// TIA Portal V17 program export: 1 tag tables, 0 data types, 3 data blocks, 1 code blocks (in call order from the OBs), 3 instance data blocks

VAR_GLOBAL   // PLC tag table "Default tag table"
   Batch_WeightScale_Done AT %M2.2 : Bool;
   Batch_FillToMixer_Done AT %M2.3 : Bool;
   Batch_Mixing_Done AT %M2.4 : Bool;
   Batch_Fillto_Pasteurisation_Done AT %M2.5 : Bool;
   Batch_Pasteurizing_Done AT %M2.6 : Bool;
   Filler_Ready AT %M2.7 : Bool;
   Clock_Byte AT %MB0 : Byte;
   Clock_10Hz AT %M0.0 : Bool;
   Clock_5Hz AT %M0.1 : Bool;
   "Clock_2.5Hz" AT %M0.2 : Bool;
   Clock_2Hz AT %M0.3 : Bool;
   "Clock_1.25Hz" AT %M0.4 : Bool;
   Clock_1Hz AT %M0.5 : Bool;
   "Clock_0.625Hz" AT %M0.6 : Bool;
   "Clock_0.5Hz" AT %M0.7 : Bool;
END_VAR

DATA_BLOCK "Device"   // DB1
{ S7_Optimized_Access := 'FALSE' }
VERSION : 0.1
// stored: AutoNumber true, DBAccessibleFromOPCUA true, DBAccessibleFromWebserver true, IsOnlyStoredInLoadMemory false, IsWriteProtectedInAS false
   VAR
      V1103 : Bool;
      V01101 : Bool;
      V2101 : Bool;
      V3101 : Bool;
      V1102 : Bool;
      V2102 : Bool;
      V3102 : Bool;
      V4101 : Bool;
      V4102 : Bool;
      V4103 : Bool;
      W1111 : Real;
      W2111 : Real;
      W3111 : Real;
      L4141 : Real;
      AGR5101 : Bool;
      PUMP4121 : Bool;
      PASTEURISING_MACHINE_ON : Bool;
      FILLING_MACHINE : Bool;
      V1101 : Bool;
      L5141 : Real;
      V01101_s : Bool;
      V2101_s : Bool;
      V3101_s : Bool;
      V1102_s : Bool;
      V2102_s : Bool;
      V3102_s : Bool;
      AGR5101_s : Bool;
      V4101_s : Bool;
      PUMP4121_s : Bool;
      V4102_s : Bool;
      PASTEURISING_MACHINE_ON_s : Bool;
      FILLING_MACHINE_s : Bool;
      V2102_ss : Bool;
      V4103_s : Bool;
   END_VAR
BEGIN
END_DATA_BLOCK

DATA_BLOCK "Recipe_Parameter"   // DB2
{ S7_Optimized_Access := 'FALSE' }
VERSION : 0.1
// stored: AutoNumber true, DBAccessibleFromOPCUA true, DBAccessibleFromWebserver true, IsOnlyStoredInLoadMemory false, IsWriteProtectedInAS false
   VAR
      SelectedFlavor : Int;
      Milk_Volume : Real;
      Flavor_Volume : Real;
      Mixing_Time : Time;
      Pasteurising_Time : Time;
   END_VAR
BEGIN
END_DATA_BLOCK

DATA_BLOCK "SCADA"   // DB3
{ S7_Optimized_Access := 'FALSE' }
VERSION : 0.1
// stored: AutoNumber true, DBAccessibleFromOPCUA true, DBAccessibleFromWebserver true, IsOnlyStoredInLoadMemory false, IsWriteProtectedInAS false
   VAR
      AutoOn : Bool;
      Start : Bool;
   END_VAR
BEGIN
END_DATA_BLOCK

ORGANIZATION_BLOCK "Main"   // OB1, LAD, ProgramCycle
TITLE = "Main Program Sweep (Cycle)"
{ S7_Optimized_Access := 'TRUE' }
VERSION : 0.1
// stored: AutoNumber true, IsIECCheckEnabled false, SetENOAutomatically false
   VAR_INPUT
      Initial_Call : Bool;   // Initial call of this OB
      Remanence : Bool;   // =True, if remanent data are available
   END_VAR
   VAR_TEMP
      "Auto/Manual" : Bool;
   END_VAR
   VAR_TEMP   // added for the SCL form of the ladder/FBD networks
      _w1 : Bool;
   END_VAR
BEGIN

REGION Network 1
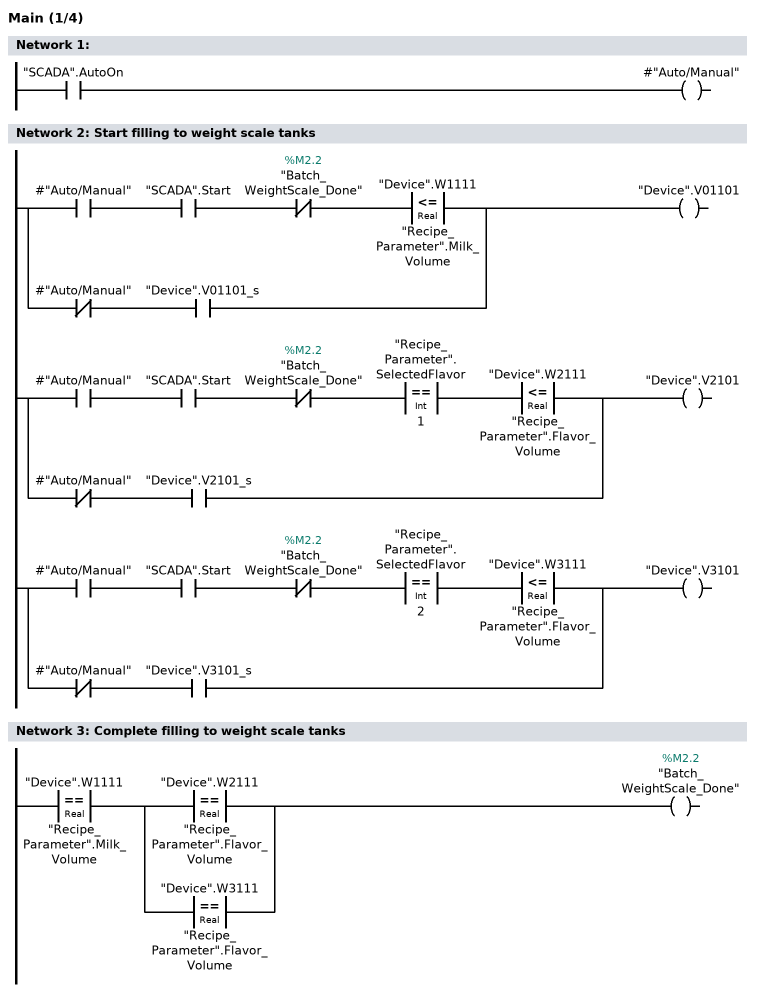
   RUNG wire#powerrail
      Contact( "SCADA".AutoOn )
      Coil( #"Auto/Manual" )
   END_RUNG
   // the same network as SCL:
   #"Auto/Manual" := "SCADA".AutoOn;
END_REGION

REGION Network 2: Start filling to weight scale tanks
   RUNG wire#powerrail
      Contact( #"Auto/Manual" )
      Contact( "SCADA".Start )
      I_Contact( "Batch_WeightScale_Done" )
      { S7_Templates := "SrcType := Real" } LE_Contact(in1 := "Device".W1111, in2 := "Recipe_Parameter".Milk_Volume)
      wire#w1
      Coil( "Device".V01101 )
   END_RUNG
   RUNG wire#powerrail
      I_Contact( #"Auto/Manual" )
      Contact( "Device".V01101_s )
   END_RUNG wire#w1
   RUNG wire#powerrail
      Contact( #"Auto/Manual" )
      Contact( "SCADA".Start )
      I_Contact( "Batch_WeightScale_Done" )
      { S7_Templates := "SrcType := Int" } EQ_Contact(in1 := "Recipe_Parameter".SelectedFlavor, in2 := 1)
      { S7_Templates := "SrcType := Real" } LE_Contact(in1 := "Device".W2111, in2 := "Recipe_Parameter".Flavor_Volume)
      wire#w2
      Coil( "Device".V2101 )
   END_RUNG
   RUNG wire#powerrail
      I_Contact( #"Auto/Manual" )
      Contact( "Device".V2101_s )
   END_RUNG wire#w2
   RUNG wire#powerrail
      Contact( #"Auto/Manual" )
      Contact( "SCADA".Start )
      I_Contact( "Batch_WeightScale_Done" )
      { S7_Templates := "SrcType := Int" } EQ_Contact(in1 := "Recipe_Parameter".SelectedFlavor, in2 := 2)
      { S7_Templates := "SrcType := Real" } LE_Contact(in1 := "Device".W3111, in2 := "Recipe_Parameter".Flavor_Volume)
      wire#w3
      Coil( "Device".V3101 )
   END_RUNG
   RUNG wire#powerrail
      I_Contact( #"Auto/Manual" )
      Contact( "Device".V3101_s )
   END_RUNG wire#w3
   // the same network as SCL:
   "Device".V01101 := (#"Auto/Manual" AND "SCADA".Start AND NOT "Batch_WeightScale_Done" AND ("Device".W1111 <= "Recipe_Parameter".Milk_Volume)) OR (NOT #"Auto/Manual" AND "Device".V01101_s);
   "Device".V2101 := (#"Auto/Manual" AND "SCADA".Start AND NOT "Batch_WeightScale_Done" AND ("Recipe_Parameter".SelectedFlavor = 1) AND ("Device".W2111 <= "Recipe_Parameter".Flavor_Volume)) OR (NOT #"Auto/Manual" AND "Device".V2101_s);
   "Device".V3101 := (#"Auto/Manual" AND "SCADA".Start AND NOT "Batch_WeightScale_Done" AND ("Recipe_Parameter".SelectedFlavor = 2) AND ("Device".W3111 <= "Recipe_Parameter".Flavor_Volume)) OR (NOT #"Auto/Manual" AND "Device".V3101_s);
END_REGION

REGION Network 3: Complete filling to weight scale tanks
   RUNG wire#powerrail
      { S7_Templates := "SrcType := Real" } EQ_Contact(in1 := "Device".W1111, in2 := "Recipe_Parameter".Milk_Volume)
      wire#w1
      { S7_Templates := "SrcType := Real" } EQ_Contact(in1 := "Device".W2111, in2 := "Recipe_Parameter".Flavor_Volume)
      wire#w2
      Coil( "Batch_WeightScale_Done" )
   END_RUNG
   RUNG wire#w1
      { S7_Templates := "SrcType := Real" } EQ_Contact(in1 := "Device".W3111, in2 := "Recipe_Parameter".Flavor_Volume)
   END_RUNG wire#w2
   // the same network as SCL:
   "Batch_WeightScale_Done" := ("Device".W1111 = "Recipe_Parameter".Milk_Volume) AND (("Device".W2111 = "Recipe_Parameter".Flavor_Volume) OR ("Device".W3111 = "Recipe_Parameter".Flavor_Volume));
END_REGION

REGION Network 4: Start filling the mixer
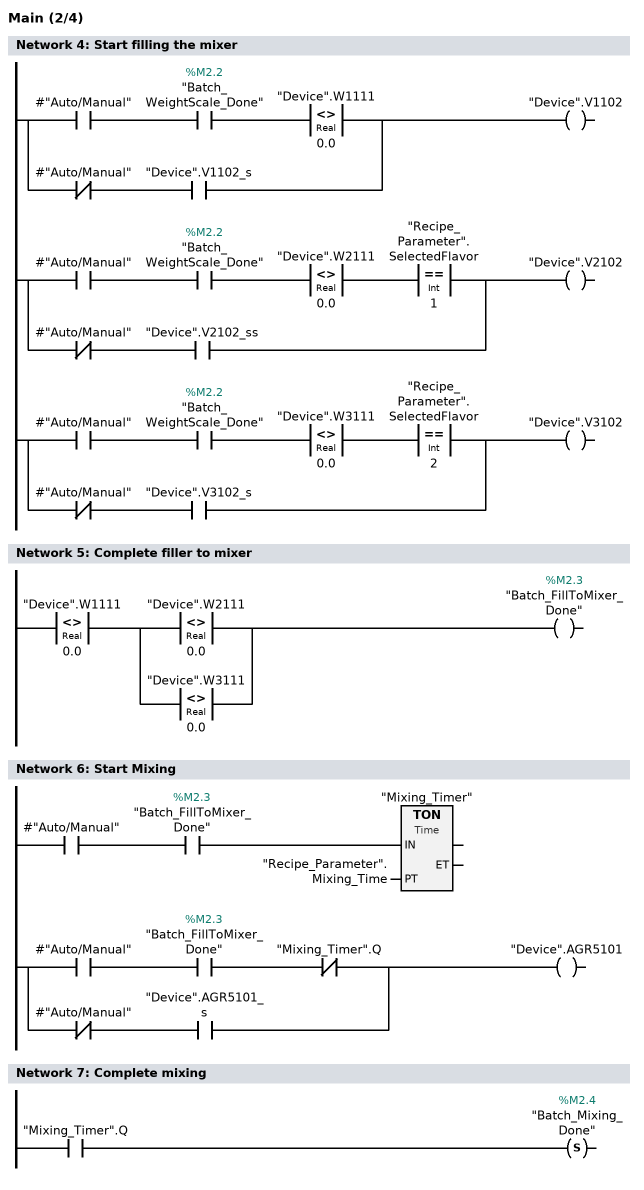
   RUNG wire#powerrail
      Contact( #"Auto/Manual" )
      Contact( "Batch_WeightScale_Done" )
      { S7_Templates := "SrcType := Real" } NE_Contact(in1 := "Device".W1111, in2 := 0.0)
      wire#w1
      Coil( "Device".V1102 )
   END_RUNG
   RUNG wire#powerrail
      I_Contact( #"Auto/Manual" )
      Contact( "Device".V1102_s )
   END_RUNG wire#w1
   RUNG wire#powerrail
      Contact( #"Auto/Manual" )
      Contact( "Batch_WeightScale_Done" )
      { S7_Templates := "SrcType := Real" } NE_Contact(in1 := "Device".W2111, in2 := 0.0)
      { S7_Templates := "SrcType := Int" } EQ_Contact(in1 := "Recipe_Parameter".SelectedFlavor, in2 := 1)
      wire#w2
      Coil( "Device".V2102 )
   END_RUNG
   RUNG wire#powerrail
      I_Contact( #"Auto/Manual" )
      Contact( "Device".V2102_ss )
   END_RUNG wire#w2
   RUNG wire#powerrail
      Contact( #"Auto/Manual" )
      Contact( "Batch_WeightScale_Done" )
      { S7_Templates := "SrcType := Real" } NE_Contact(in1 := "Device".W3111, in2 := 0.0)
      { S7_Templates := "SrcType := Int" } EQ_Contact(in1 := "Recipe_Parameter".SelectedFlavor, in2 := 2)
      wire#w3
      Coil( "Device".V3102 )
   END_RUNG
   RUNG wire#powerrail
      I_Contact( #"Auto/Manual" )
      Contact( "Device".V3102_s )
   END_RUNG wire#w3
   // the same network as SCL:
   "Device".V1102 := (#"Auto/Manual" AND "Batch_WeightScale_Done" AND ("Device".W1111 <> 0.0)) OR (NOT #"Auto/Manual" AND "Device".V1102_s);
   "Device".V2102 := (#"Auto/Manual" AND "Batch_WeightScale_Done" AND ("Device".W2111 <> 0.0) AND ("Recipe_Parameter".SelectedFlavor = 1)) OR (NOT #"Auto/Manual" AND "Device".V2102_ss);
   "Device".V3102 := (#"Auto/Manual" AND "Batch_WeightScale_Done" AND ("Device".W3111 <> 0.0) AND ("Recipe_Parameter".SelectedFlavor = 2)) OR (NOT #"Auto/Manual" AND "Device".V3102_s);
END_REGION

REGION Network 5: Complete filler to mixer
   RUNG wire#powerrail
      { S7_Templates := "SrcType := Real" } NE_Contact(in1 := "Device".W1111, in2 := 0.0)
      wire#w1
      { S7_Templates := "SrcType := Real" } NE_Contact(in1 := "Device".W2111, in2 := 0.0)
      wire#w2
      Coil( "Batch_FillToMixer_Done" )
   END_RUNG
   RUNG wire#w1
      { S7_Templates := "SrcType := Real" } NE_Contact(in1 := "Device".W3111, in2 := 0.0)
   END_RUNG wire#w2
   // the same network as SCL:
   "Batch_FillToMixer_Done" := ("Device".W1111 <> 0.0) AND (("Device".W2111 <> 0.0) OR ("Device".W3111 <> 0.0));
END_REGION

REGION Network 6: Start Mixing
   RUNG wire#powerrail
      Contact( #"Auto/Manual" )
      Contact( "Batch_FillToMixer_Done" )
      { S7_Templates := "time_type := Time" } "Mixing_Timer".TON(pt := "Recipe_Parameter".Mixing_Time, et =>)
   END_RUNG
   RUNG wire#powerrail
      Contact( #"Auto/Manual" )
      Contact( "Batch_FillToMixer_Done" )
      I_Contact( "Mixing_Timer".Q )
      wire#w1
      Coil( "Device".AGR5101 )
   END_RUNG
   RUNG wire#powerrail
      I_Contact( #"Auto/Manual" )
      Contact( "Device".AGR5101_s )
   END_RUNG wire#w1
   // the same network as SCL:
   "Mixing_Timer".TON(IN := #"Auto/Manual" AND "Batch_FillToMixer_Done", PT := "Recipe_Parameter".Mixing_Time);
   "Device".AGR5101 := (#"Auto/Manual" AND "Batch_FillToMixer_Done" AND NOT "Mixing_Timer".Q) OR (NOT #"Auto/Manual" AND "Device".AGR5101_s);
END_REGION

REGION Network 7: Complete mixing
   RUNG wire#powerrail
      Contact( "Mixing_Timer".Q )
      S_Coil( "Batch_Mixing_Done" )
   END_RUNG
   // the same network as SCL:
   IF "Mixing_Timer".Q THEN "Batch_Mixing_Done" := TRUE; END_IF;
END_REGION

REGION Network 8: Start filling to pasteurising machine
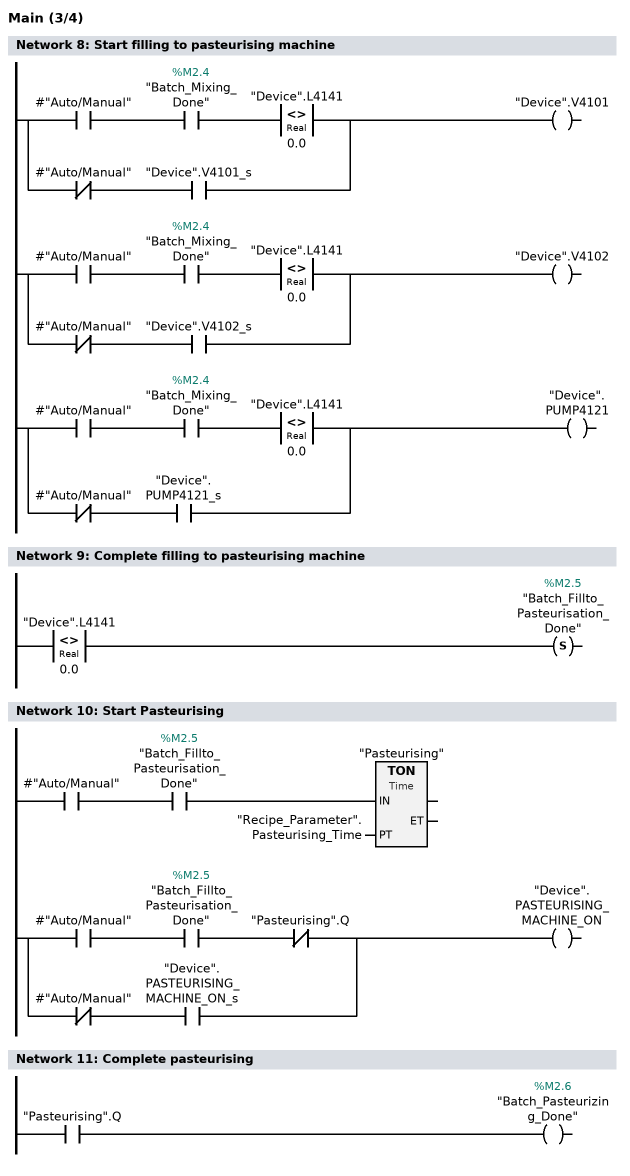
   RUNG wire#powerrail
      Contact( #"Auto/Manual" )
      Contact( "Batch_Mixing_Done" )
      { S7_Templates := "SrcType := Real" } NE_Contact(in1 := "Device".L4141, in2 := 0.0)
      wire#w1
      Coil( "Device".V4101 )
   END_RUNG
   RUNG wire#powerrail
      I_Contact( #"Auto/Manual" )
      Contact( "Device".V4101_s )
   END_RUNG wire#w1
   RUNG wire#powerrail
      Contact( #"Auto/Manual" )
      Contact( "Batch_Mixing_Done" )
      { S7_Templates := "SrcType := Real" } NE_Contact(in1 := "Device".L4141, in2 := 0.0)
      wire#w2
      Coil( "Device".V4102 )
   END_RUNG
   RUNG wire#powerrail
      I_Contact( #"Auto/Manual" )
      Contact( "Device".V4102_s )
   END_RUNG wire#w2
   RUNG wire#powerrail
      Contact( #"Auto/Manual" )
      Contact( "Batch_Mixing_Done" )
      { S7_Templates := "SrcType := Real" } NE_Contact(in1 := "Device".L4141, in2 := 0.0)
      wire#w3
      Coil( "Device".PUMP4121 )
   END_RUNG
   RUNG wire#powerrail
      I_Contact( #"Auto/Manual" )
      Contact( "Device".PUMP4121_s )
   END_RUNG wire#w3
   // the same network as SCL:
   "Device".V4101 := (#"Auto/Manual" AND "Batch_Mixing_Done" AND ("Device".L4141 <> 0.0)) OR (NOT #"Auto/Manual" AND "Device".V4101_s);
   "Device".V4102 := (#"Auto/Manual" AND "Batch_Mixing_Done" AND ("Device".L4141 <> 0.0)) OR (NOT #"Auto/Manual" AND "Device".V4102_s);
   "Device".PUMP4121 := (#"Auto/Manual" AND "Batch_Mixing_Done" AND ("Device".L4141 <> 0.0)) OR (NOT #"Auto/Manual" AND "Device".PUMP4121_s);
END_REGION

REGION Network 9: Complete filling to pasteurising machine
   RUNG wire#powerrail
      { S7_Templates := "SrcType := Real" } NE_Contact(in1 := "Device".L4141, in2 := 0.0)
      S_Coil( "Batch_Fillto_Pasteurisation_Done" )
   END_RUNG
   // the same network as SCL:
   IF "Device".L4141 <> 0.0 THEN "Batch_Fillto_Pasteurisation_Done" := TRUE; END_IF;
END_REGION

REGION Network 10: Start Pasteurising
   RUNG wire#powerrail
      Contact( #"Auto/Manual" )
      Contact( "Batch_Fillto_Pasteurisation_Done" )
      { S7_Templates := "time_type := Time" } "Pasteurising".TON(pt := "Recipe_Parameter".Pasteurising_Time, et =>)
   END_RUNG
   RUNG wire#powerrail
      Contact( #"Auto/Manual" )
      Contact( "Batch_Fillto_Pasteurisation_Done" )
      I_Contact( "Pasteurising".Q )
      wire#w1
      Coil( "Device".PASTEURISING_MACHINE_ON )
   END_RUNG
   RUNG wire#powerrail
      I_Contact( #"Auto/Manual" )
      Contact( "Device".PASTEURISING_MACHINE_ON_s )
   END_RUNG wire#w1
   // the same network as SCL:
   "Pasteurising".TON(IN := #"Auto/Manual" AND "Batch_Fillto_Pasteurisation_Done",
                      PT := "Recipe_Parameter".Pasteurising_Time);
   "Device".PASTEURISING_MACHINE_ON := (#"Auto/Manual" AND "Batch_Fillto_Pasteurisation_Done" AND NOT "Pasteurising".Q) OR (NOT #"Auto/Manual" AND "Device".PASTEURISING_MACHINE_ON_s);
END_REGION

REGION Network 11: Complete pasteurising
   RUNG wire#powerrail
      Contact( "Pasteurising".Q )
      Coil( "Batch_Pasteurizing_Done" )
   END_RUNG
   // the same network as SCL:
   "Batch_Pasteurizing_Done" := "Pasteurising".Q;
END_REGION

REGION Network 12: Start filling to filling machine, after 5s will be ready to fill the bottles
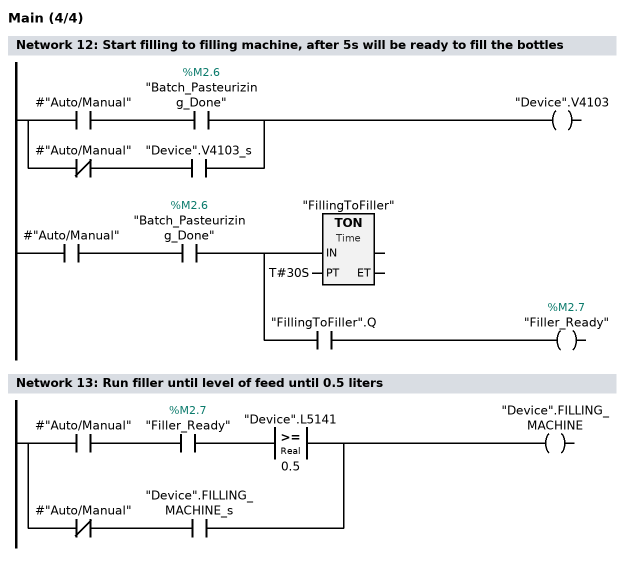
   RUNG wire#powerrail
      Contact( #"Auto/Manual" )
      Contact( "Batch_Pasteurizing_Done" )
      wire#w1
      Coil( "Device".V4103 )
   END_RUNG
   RUNG wire#powerrail
      I_Contact( #"Auto/Manual" )
      Contact( "Device".V4103_s )
   END_RUNG wire#w1
   RUNG wire#powerrail
      Contact( #"Auto/Manual" )
      Contact( "Batch_Pasteurizing_Done" )
      wire#w2
      { S7_Templates := "time_type := Time" } "FillingToFiller".TON(pt := T#30S, et =>)
   END_RUNG
   RUNG wire#w2
      Contact( "FillingToFiller".Q )
      Coil( "Filler_Ready" )
   END_RUNG
   // the same network as SCL:
   "Device".V4103 := (#"Auto/Manual" AND "Batch_Pasteurizing_Done") OR (NOT #"Auto/Manual" AND "Device".V4103_s);
   #_w1 := #"Auto/Manual" AND "Batch_Pasteurizing_Done";
   "FillingToFiller".TON(IN := #_w1, PT := T#30S);
   "Filler_Ready" := #_w1 AND "FillingToFiller".Q;
END_REGION

REGION Network 13: Run filler until level of feed until 0.5 liters
   RUNG wire#powerrail
      Contact( #"Auto/Manual" )
      Contact( "Filler_Ready" )
      { S7_Templates := "SrcType := Real" } GE_Contact(in1 := "Device".L5141, in2 := 0.5)
      wire#w1
      Coil( "Device".FILLING_MACHINE )
   END_RUNG
   RUNG wire#powerrail
      I_Contact( #"Auto/Manual" )
      Contact( "Device".FILLING_MACHINE_s )
   END_RUNG wire#w1
   // the same network as SCL:
   "Device".FILLING_MACHINE := (#"Auto/Manual" AND "Filler_Ready" AND ("Device".L5141 >= 0.5)) OR (NOT #"Auto/Manual" AND "Device".FILLING_MACHINE_s);
END_REGION
END_ORGANIZATION_BLOCK

DATA_BLOCK "FillingToFiller"   // DB4
{ S7_Optimized_Access := 'TRUE' }
// stored: AutoNumber true, DBAccessibleFromOPCUA true, DBAccessibleFromWebserver true, InstanceOfName IEC_TIMER, OfSystemLibElement IEC_TIMER, OfSystemLibVersion 1.0
"IEC_TIMER"
   // VAR
   //    PT : Time;
   //    ET { ExternalWritable := 'False'} : Time;
   //    IN : Bool;
   //    Q { ExternalWritable := 'False'} : Bool;
   // END_VAR
BEGIN
END_DATA_BLOCK

DATA_BLOCK "Mixing_Timer"   // DB5
{ S7_Optimized_Access := 'TRUE' }
// stored: AutoNumber true, DBAccessibleFromOPCUA true, DBAccessibleFromWebserver true, InstanceOfName IEC_TIMER, OfSystemLibElement IEC_TIMER, OfSystemLibVersion 1.0
"IEC_TIMER"
   // VAR
   //    PT : Time;
   //    ET { ExternalWritable := 'False'} : Time;
   //    IN : Bool;
   //    Q { ExternalWritable := 'False'} : Bool;
   // END_VAR
BEGIN
END_DATA_BLOCK

DATA_BLOCK "Pasteurising"   // DB6
{ S7_Optimized_Access := 'TRUE' }
// stored: AutoNumber true, DBAccessibleFromOPCUA true, DBAccessibleFromWebserver true, InstanceOfName IEC_TIMER, OfSystemLibElement IEC_TIMER, OfSystemLibVersion 1.0
"IEC_TIMER"
   // VAR
   //    PT : Time;
   //    ET { ExternalWritable := 'False'} : Time;
   //    IN : Bool;
   //    Q { ExternalWritable := 'False'} : Bool;
   // END_VAR
BEGIN
END_DATA_BLOCK
